FUNCTION_BLOCK FB_SAVE_1D (* Stores 1 min resolved data in a 1 day array *)
  (* Standard: 61499-2 *)
  (* Version 1.0, 2017-09-01, Marc Jakobi, HTW Berlin *)
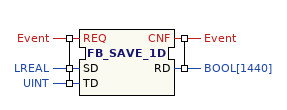
  EVENT_INPUT
    REQ WITH SD, TD; (* Normal Execution Request *)
  END_EVENT
  EVENT_OUTPUT
    CNF WITH RD; (* Execution Confirmation *)
  END_EVENT
  VAR_INPUT
    SD : LREAL; (* Data to be stored *)
    TD : UINT; (* Time of day [0, ..,1339] *)
  END_VAR
  VAR_OUTPUT
    RD : ARRAY [0..1439] OF BOOL; (* Array containing 1 day of stored data *)
  END_VAR
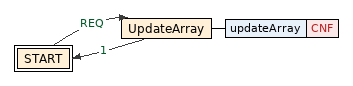
  EC_STATES
    START; (* Initial State *)
    UpdateArray : updateArray -> CNF; (* Normal execution *)
  END_STATES
  EC_TRANSITIONS
    START TO UpdateArray := REQ;
    UpdateArray TO START := 1;
  END_TRANSITIONS
  ALGORITHM updateArray IN ST: (* Updates the output array with the incoming data. *)
RD[TD] := SD;
  END_ALGORITHM
END_FUNCTION_BLOCK
